(* CoDeSys 2.3.9.41 project: Coffee_Maker.pro *)
(* Libraries: Standard.lib 4.10.05 11:14:46, IecSfc.lib 13.4.06 15:51:28, SYSLIBCALLBACK.LIB 26.9.08 16:43:52 *)

(* Task configuration *)
TASK NewTask (PRIORITY := 1); (* freewheeling *)
	VIS_PRG();
	PLC_Timers();
	PLC_ST_PRG();
END_TASK

(* Global variable list: Global_Variables *)
VAR_GLOBAL
(* Счётчики Counters -- префикс ctr *)
	ctrPrtn: UINT := 0;	(*счётчик порций кофе*)
(* Входы *)
	(* Кнопки Push Buttons -- префикс pb *)
	pbStart: BOOL;	(*Кнопка "Пуск"*)
	pbStop: BOOL;	(*Кнопка "Заверш"*)
	pbEmStop: BOOL;	(*Кнопка "Авост"*)
	pbPlus, _pbPlus: BOOL;	(*Кнопка "Плюс"*)
	pbMinus, _pbMinus: BOOL;	(*Кнопка "Минус"*)
	 (* Датчики Sensors -- префикс s *)
	sUT: BOOL;	(* датчик верхней температуры нагревателя*)
	sLT: BOOL;	(* датчик нижней температуры нагревателя*)
	sWT, _sWT: BOOL;	(* датчик рабочей температуры нагревателя*)
	sWL: BOOL;	(* датчик уровня воды*)
(*Выходы*)
	(* Клапаны/Лампы Valves/Lamps -- префикс vlv/lmp *)
	vlv1, _vlv1: BOOL;        (* открыть клапан 1*)
	vlv2, _vlv2: BOOL;        (* открыть клапан 2 *)
	(* Приводы/Лампы Actuators/Lamps -- префикс act/lmp*)
 	actHtr, _actHtr: BOOL;    (* включить нагреватель*)
    	(* Режимы/Состояния/Лампы Modes/States/Lamps -- префикс m/q/lmp *)
	mWtrSup, _mWtrSup: BOOL;	(*подача воды*)
	mStmRel, _mStmRel: BOOL;	(*выпуск пара*)
	mHeat, _mHeat: BOOL;	(*нагревание/кипячение*)
	mSysOn,  _mSysOn : BOOL;  (* система включена                               *)
	mCompl,  _mCompl : BOOL;  (* режим плавного завершения работы установки     *)
	mEmStop, _mEmStop: BOOL;	(*аварийная остановка*)
	(* Ошибки/Лампы Errors/Lamps -- префикс err/lmp *)
	errHtr, _errHtr: BOOL;    (* сигнал ошибки нагревателя                      *)
	(*Псевдодатчики/Лампы Pseudosensors/Lamps -- префикс ps/lmp*)
	psL0, _psL0: BOOL;	(*уровень 0 в ёмкости*)
	psL1, _psL1: BOOL;	(*уровень 1 в ёмкости*)
	psStmPr, _psStmPr: BOOL;	(*пар/давление в ёмкости*)
	(* Дисплей Display -- префикс d *)
	dBit0: BOOL;
	dBit1: BOOL;
	dBit2: BOOL;
(* Вспомогательные переменные Conditions -- префикс c *)
	cFin: BOOL;               (* условие завершения работы кофеварки            *)
(* Таймеры Timers -- префикс tmr *)
	tmrHtr: TON := (PT := T#12s);	(*таймер ожидания нагрева*)
	tmrWtr: TON := (PT := T#2s);	(*таймер подачи воды*)
	tmrStm: TON := (PT := T#2s);	(*таймер выпуска пара*)
	tmrHeat: TON := (PT := T#5s);	(*таймер нагрева воды*)
END_VAR

(* POU VIS_PRG, ST *)
PROGRAM VIS_PRG
VAR
	(* ------- Обычные кнопки ------- *)
	PBTnk: BOOL;	(* наполнить резервуар водой *)
	PBCmp: BOOL;	(* осушить резервуар с водой *)
	(* ------- Кнопки-переключатели ------- *)
	SBHtrBrk: BOOL;	(* поломка нагревателя *)
	(* ------- Жидкости ------- *)
	Wtr, _Wtr: INT;	(* объём воды в резервуаре *)
	Stm, _Stm: INT;	(* объём воды в ёмкости для кипячения *)
	Cof, _Cof: INT;	(* объём кофе *)
	WtrClr: DWORD:=16#00_FF_80_00;	(* температура воды в ёмкости для нагревателя *)
	WtrBlue, _WtrBlue: BYTE;	(* степень нагрева воды *)
	(* ------- Нагреватель ------- *)
  	HtrClr: DWORD:=16#00_FF_FF_FF; (* температура нагревателя (цвет)         *)
  	HtrRed, _HtrRed: BYTE;         (* степень накаливания нагревателя        *)
  	HtrOn: BOOL;                   (* нагреватель функционирует (греет)      *)
END_VAR
Wtr:= MAX(0,MIN(460,BOOL_TO_INT(NOT PBCmp)*_Wtr+BOOL_TO_INT(PBTnk)*460-BOOL_TO_INT(vlv1)));
Stm:= MAX(0,_Stm+BOOL_TO_INT(vlv1 AND _Wtr>30)-BOOL_TO_INT(vlv2 AND _Stm>0));
Cof:= MAX(0,_Cof+BOOL_TO_INT(vlv2 AND Stm>0));
WtrBlue:=_WtrBlue+BOOL_TO_BYTE(tmrHeat.IN AND _WtrBlue<255)-BOOL_TO_BYTE(mEmStop AND NOT mHeat AND NOT psStmPr AND _WtrBlue>0);
IF NOT psL0 THEN WtrBlue:=0; END_IF
WtrClr:=65536*255+256*(128+WtrBlue*3/2)+WtrBlue*3/2;
(* ------- Нагреватель ------- *)
HtrOn:=actHtr AND NOT SBHtrBrk; (* нагреватель включается, если не сломан       *)
HtrRed:=_HtrRed+BOOL_TO_BYTE(HtrOn AND _HtrRed<255)-BOOL_TO_BYTE(NOT HtrOn AND _HtrRed>0);
HtrClr:=65536*(255-HtrRed)+256*(255-HtrRed)+255;
(* ------- Выставление сигналов датчиков ------- *)
sWL:=(Wtr>30);
sUT:=(HtrRed>=252);
sLT:=(HtrRed>=160);
sWT:=(HtrRed>=150);
(* -------  Псевдооператорный раздел ------- *)
_Wtr:= Wtr; _Stm:=Stm; _Cof:= Cof; _HtrRed:=HtrRed; _WtrBlue:=WtrBlue;
END_PROGRAM

(* POU PLC_Timers, FBD *)
PROGRAM PLC_Timers
VAR
END_VAR
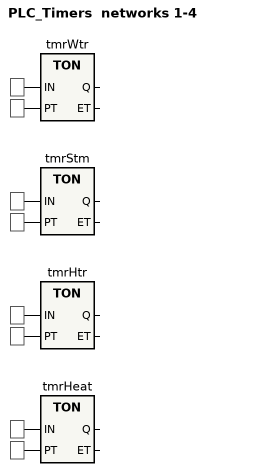
_FBD_ (* Function Block Diagram *)
NETWORK 1
	tmrWtr:TON(IN: , PT: )
NETWORK 2
	tmrStm:TON(IN: , PT: )
NETWORK 3
	tmrHtr:TON(IN: , PT: )
NETWORK 4
	tmrHeat:TON(IN: , PT: )
_END_FBD_
END_PROGRAM

(* POU PLC_ST_PRG, ST *)
PROGRAM PLC_ST_PRG
VAR
END_VAR
(* ------- Счётчики ------- *)
IF NOT _pbPlus AND pbPlus AND ctrPrtn < 7 THEN	(* ctrPrtn+1 *)
    ctrPrtn := ctrPrtn + 1;
END_IF;
IF NOT _pbMinus AND pbMinus AND ctrPrtn > 0 AND NOT _psL0 THEN	(* ctrPrtn-1 *)
    ctrPrtn := ctrPrtn - 1;
END_IF;
IF pbEmStop THEN	(* ctrPrtn:=0 *)
    ctrPrtn := 0;
END_IF;
IF NOT _pbMinus AND tmrStm.Q AND NOT _mEmStop AND ctrPrtn > 0 THEN	(* ctrPrtn-1 *)
    ctrPrtn := ctrPrtn - 1;
END_IF;
(* ------- Дисплей ------- *)
dBit0 := ctrPrtn.0;  (* dBit0 *)
dBit1 := ctrPrtn.1;  (* dBit1 *)
dBit2 := ctrPrtn.2;  (* dBit2 *)
(* ------- Ошибки/Лампы ------- *)
IF NOT _errHtr AND NOT sWT AND (tmrHtr.Q OR _actHtr AND _sWT) THEN errHtr:=1;         (* errHtr+  *)
ELSIF  _errHtr AND pbEmStop                                     THEN errHtr:=0;         (* errHtr-  *)
END_IF;
(* ------- Псевдодатчики/Лампы ------- *)
IF NOT _psL0 AND _vlv1 	THEN psL0 := 1;	(* psL0+ *)
ELSIF _psL0 AND tmrStm.Q THEN psL0 := 0;	(* psL0- *)
END_IF;
IF NOT _psL1 AND tmrWtr.Q THEN psL1 := 1;	(* psL1+ *)
ELSIF _psL1 AND _mStmRel THEN psL1 := 0;	(* psL1- *)
END_IF;
IF NOT _psStmPr AND psL0 AND tmrHeat.Q THEN psStmPr := 1;	(* psStmPr+ *)
ELSIF _psStmPr AND NOT psL0 THEN psStmPr := 0;	(* psStmPr- *)
END_IF;
(* ------- Вспомогательные переменные ------- *)
cFin := pbEmStop OR errHtr OR
		NOT psL0 AND _mCompl OR
		ctrPrtn = 0 OR NOT sWL;	(* cFin *)
(* ------- Режимы/Состояния/Лампы ------- *)
IF NOT _mSysOn AND pbStart AND NOT cFin THEN mSysOn:=1;	(* mSysOn+  *)
ELSIF  _mSysOn AND                cFin THEN mSysOn:=0;	(* mSysOn-  *)
END_IF;
IF NOT _mCompl AND     mSysOn AND pbStop THEN mCompl:=1;	(* mCompl+  *)
ELSIF  _mCompl AND NOT mSysOn            THEN mCompl:=0;		(* mCompl-  *)
END_IF;
IF NOT _mEmStop AND pbEmStop AND psL0 THEN mEmStop := 1;	(* mEmStop+ *)
ELSIF _mEmStop AND NOT psL0 THEN mEmStop := 0;	(* mEmStop- *)
END_IF;
IF NOT _mWtrSup AND mSysOn AND NOT psL0 THEN mWtrSup := 1;	(* mWtrSup+ *)
ELSIF _mWtrSup AND (NOT mSysOn OR psL1) THEN mWtrSup := 0;	(* mWtrSup- *)
END_IF;
IF NOT _mHeat AND mSysOn AND NOT psStmPr AND (psL1 OR mEmStop) THEN mHeat := 1;	(* mHeat+ *)
ELSIF _mHeat AND (NOT mSysOn OR psStmPr) THEN mHeat := 0;	(* mHeat- *)
END_IF;
IF NOT _mStmRel AND mSysOn AND psStmPr THEN mStmRel := 1;	(* mStmRel+ *)
ELSIF _mStmRel AND (NOT mSysOn OR NOT psStmPr) THEN mStmRel := 0;	(* mStmRel- *)
END_IF;
(* ------- Нагреватель/Лампа ------- *)
IF NOT _actHtr AND      mSysOn AND NOT sLT  THEN actHtr:=1;                           (* actHtr+  *)
ELSIF  _actHtr AND (NOT mSysOn OR      sUT) THEN actHtr:=0;                           (* actHtr-  *)
END_IF;
(* ------- Клапаны/Приводы/Лампы ------- *)
vlv1 := tmrWtr.IN;	(* vlv1 *)
vlv2 := tmrStm.IN;	(* vlv2 *)
(* ------- Раздел таймеров ------- *)
tmrHtr.IN := actHtr AND NOT sWT;	(* tmrHtr.IN *)
tmrWtr.IN := sWL AND mWtrSup;	(* tmrWtr.IN *)
tmrStm.IN := mStmRel;	(* tmrStm.IN *)
tmrHeat.IN := sWT AND mHeat;	(* tmrHeat.IN *)
(* ------- Псевдооператорный раздел ------- *)
_errHtr:=errHtr; _psL0:= psL0; _psL1:= psL1;
_psStmPr:=psStmPr; _mSysOn:=mSysOn; _mCompl:=MCompl;
_mEmStop:=mEmStop; _mWtrSup:=mWtrSup; _mHeat:=mHeat;
_mStmRel:=mStmRel; _actHtr:=actHtr; _sWT:=sWT;
_vlv1:=vlv1; _vlv2:=vlv2; _pbPlus:=pbPlus; _pbMinus:=pbMinus;
END_PROGRAM

(* Visualisation VIS_CoffeeMaker
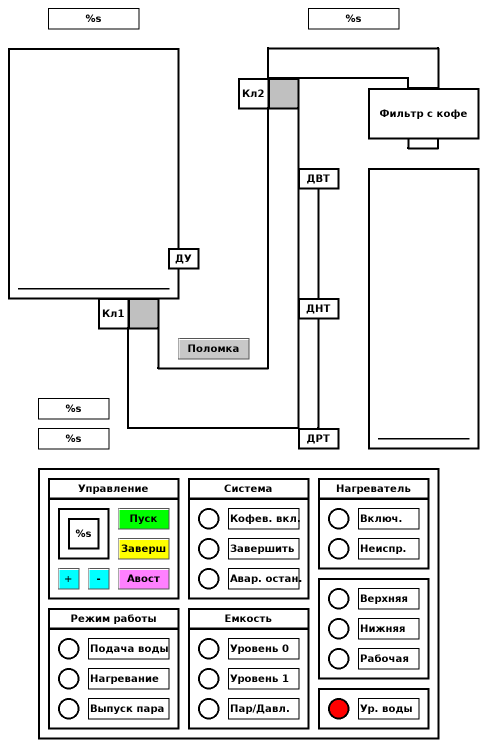
rectangle at (70,490)-(201,511): text "Управление"
button at (140,520)-(191,541): text "Пуск"; taps .pbStart
button at (140,550)-(191,571): text "Заверш"; taps .pbStop
button at (140,580)-(191,601): text "Авост"; taps .pbEmStop
rectangle at (70,620)-(201,641): text "Режим работы"
button at (80,580)-(101,601): text "+"; taps .pbPlus
button at (110,580)-(131,601): text "-"; taps .pbMinus
ellipse at (80,650)-(101,671): alarm colour if .mWtrSup
ellipse at (80,680)-(101,701): alarm colour if .mHeat
ellipse at (80,710)-(101,731): alarm colour if .mStmRel
rectangle at (110,650)-(191,671): text "Подача воды"
rectangle at (110,680)-(191,701): text "Нагревание"
rectangle at (110,710)-(191,731): text "Выпуск пара"
rectangle at (210,490)-(331,511): text "Система"
ellipse at (220,520)-(241,541): alarm colour if .mSysOn
ellipse at (220,550)-(241,571): alarm colour if .mCompl
ellipse at (220,580)-(241,601): alarm colour if .mEmStop
rectangle at (250,520)-(321,541): text "Кофев. вкл."
rectangle at (250,550)-(321,571): text "Завершить"
rectangle at (250,580)-(321,601): text "Авар. остан."
rectangle at (210,620)-(331,641): text "Емкость"
ellipse at (220,650)-(241,671): alarm colour if .psL0
ellipse at (220,680)-(241,701): alarm colour if .psL1
ellipse at (220,710)-(241,731): alarm colour if .psStmPr
rectangle at (250,650)-(321,671): text "Уровень 0"
rectangle at (250,680)-(321,701): text "Уровень 1"
rectangle at (250,710)-(321,731): text "Пар/Давл."
rectangle at (340,490)-(451,511): text "Нагреватель"
ellipse at (350,520)-(371,541): alarm colour if .actHtr
ellipse at (350,550)-(371,571): alarm colour if .errHtr
ellipse at (350,600)-(371,621): alarm colour if .sUT
ellipse at (350,630)-(371,651): alarm colour if .sLT
ellipse at (350,660)-(371,681): alarm colour if .sWT
ellipse at (350,710)-(371,731): alarm colour if .sWL
rectangle at (380,520)-(441,541): text "Включ."
rectangle at (380,550)-(441,571): text "Неиспр."
rectangle at (380,600)-(441,621): text "Верхняя"
rectangle at (380,630)-(441,651): text "Нижняя"
rectangle at (380,660)-(441,681): text "Рабочая"
rectangle at (380,710)-(441,731): text "Ур. воды"
rectangle at (90,530)-(121,561): text "%s"; shows .ctrPrtn
rectangle at (390,100)-(501,151): text "Фильтр с кофе"
rectangle at (320,180)-(361,201): text "ДВТ"; alarm colour if .sUT
rectangle at (320,310)-(361,331): text "ДНТ"; alarm colour if .sLT
rectangle at (320,440)-(361,461): text "ДРТ"; alarm colour if .sWT
rectangle at (150,310)-(181,341): alarm colour if .vlv1
rectangle at (120,310)-(151,341): text "Кл1"; alarm colour if .vlv1
rectangle at (290,90)-(321,121): alarm colour if .vlv2
rectangle at (260,90)-(291,121): text "Кл2"; alarm colour if .vlv2
rounded rectangle at (30,60)-(201,311): taps VIS_PRG.PBTnk
rectangle at (190,260)-(221,281): text "ДУ"; alarm colour if .sWL
rectangle at (70,20)-(161,41): text "%s"; shows .tmrWtr.ET
rectangle at (60,440)-(131,461): text "%s"; shows .tmrHtr.ET
rectangle at (60,410)-(131,431): text "%s"; shows .tmrHeat.ET
rectangle at (330,20)-(421,41): text "%s"; shows .tmrStm.ET
button at (200,350)-(271,371): text "Поломка"; toggles VIS_PRG.SBHtrBrk
rectangle at (40,300)-(191,301): taps VIS_PRG.PBCmp; top -VIS_PRG.Wtr/2
rectangle at (400,450)-(491,451): top -VIS_PRG.Cof
15 more shapes without text or variables
4 elements of other kinds (tables, trends, ...) not read
*)
